PROGRAM MAIN
VAR
	SerialComm	: FB_EL6001;
END_VAR

END_PROGRAM

(* stored: Version 1.1.0.1, ProductVersion 3.1.4024.9
   POU MAIN: Id {1b25311b-b9b7-4ec0-ae90-6b6dc302e5fd}, SpecialFunc None *)
